// TwinCAT 3 PLC project Untitled1
// ProgramVersion: 3.1.4026.16
// libraries:
//   Tc2_Standard, * (Beckhoff Automation GmbH)
//   Tc2_System, * (Beckhoff Automation GmbH)
// project tree:
//   / PlcTask.TcTTO
//   POUs/ MAIN.TcPOU, Rampa.TcPOU
// real-time tasks:
//   TASK PlcTask: cycle T#10ms, priority 20, ADS port 350

CONFIGURATION Untitled1
    RESOURCE PLC ON TwinCAT3
        TASK PlcTask(INTERVAL := T#10ms, PRIORITY := 20);
        PROGRAM MAIN WITH PlcTask : MAIN;
    END_RESOURCE
END_CONFIGURATION

// ---- POUs/MAIN.TcPOU
PROGRAM MAIN
VAR
	bStartButton : BOOL;
	bEmergencyStopButton : BOOL;

	fbRampaBlogu : Rampa;
	rTarget : REAL;
	rAuxTarget : REAL;
	rAccelerationTime : REAL := 4;
	rDecelerationTime : REAL := 2;
	rTargetDirectioonn : BOOL;
	rDirection : BOOL;
	
	rRPM : REAL;
	bFwStart : BOOL;
	bBwStart : BOOL;
END_VAR

IF bEmergencyStopButton THEN
	bFwStart := FALSE;
	bBwStart := FALSE;
	
	fbRampaBlogu(
	rTargetRPM:= 0,
	rInDirection:= rTargetDirectioonn, 
	rAccTime:= rAccelerationTime, 
	rDecTime:= rDecelerationTime, 
	rUpdateRPM:= TRUE, 
	rNewRPM:= 0, 
	rRPM=> rRPM,
	rCurrentDirection => rDirection);

ELSE
	IF bStartButton THEN
		rAuxTarget := rTarget;
	ELSE
		rAuxTarget := 0;
	END_IF
	
	fbRampaBlogu(
	rTargetRPM:= rAuxTarget,
	rInDirection:= rTargetDirectioonn, 
	rAccTime:= rAccelerationTime, 
	rDecTime:= rDecelerationTime, 
	rUpdateRPM:= FALSE, 
	rNewRPM:= 0, 
	rRPM=> rRPM,
	rCurrentDirection => rDirection);
END_IF

	IF rRPM = 0 THEN
		bFwStart := FALSE;
		bBwStart := FALSE;	
	ELSIF rDirection THEN
		bFwStart := FALSE;
		bBwStart := TRUE;
	ELSE
		bFwStart := TRUE;
		bBwStart := FALSE;
	END_IF

END_PROGRAM

// ---- POUs/Rampa.TcPOU
FUNCTION_BLOCK Rampa
VAR_INPUT
	rTargetRPM : REAL;
	rInDirection : BOOL;
	
	rAccTime : REAL;
	rDecTime : REAL;
	
	rUpdateRPM : BOOL;
	rNewRPM : REAL;
END_VAR
VAR_OUTPUT
	rRPM : REAL := 0;
	rCurrentDirection : BOOL;
END_VAR
VAR
	rAuxTargetRPM : REAL;
	rRampTime : REAL;
	
	rOldTargetRPM : REAL;
	rStartRPM : REAL;
	rDifference : REAL;
	rAddRPM : REAL;
	iTime : INT := 0;
END_VAR

IF rCurrentDirection <> rInDirection THEN
	rAuxTargetRPM := 0;
ELSE 
	rAuxTargetRPM := rTargetRPM;
END_IF

IF rOldTargetRPM <> rAuxTargetRPM THEN
	rOldTargetRPM := rAuxTargetRPM;
	rStartRPM := rRPM;
	iTime := 0;
END_IF

IF rRPM <> rAuxTargetRPM THEN
	rDifference := rAuxTargetRPM - rStartRPM;
	
	rRampTime := SEL(rAuxTargetRPM < rRPM, rAccTime, rDecTime);
	
	rAddRPM := rDifference * (1 - COS(((INT_TO_REAL(iTime)/100)/rRampTime)*pi*2))/2;	
	
	iTime := iTime + 1;
END_IF

IF rRPM = 0 AND rTargetRPM <> rRPM AND rCurrentDirection <> rInDirection THEN
	rCurrentDirection := rInDirection;
END_IF

rRPM := rStartRPM + rAddRPM;

IF rUpdateRPM THEN
	rRPM := rNewRPM;
	iTime := 0;
END_IF

END_FUNCTION_BLOCK
